// TIA Portal project "Template_ITIA2021" (V15.1)

(* hardware
DEVICE "S71500/ET200MP station_1"  S7-1500 station
   slot 0: "Rail_0"  Rack  6ES7 590-1***0-0AA0
   slot 0: "PM 70W 120/230VAC"  PM 70W 120/230VAC  6EP1332-4BA00
   slot 1: "Target_12_PLC"  CPU 1513-1 PN  6ES7 513-1AL02-0AB0  V2.6
      slot 3: "CPU display_1"  6ES7591-1AA00-0AA0
DEVICE "S71500/ET200MP station_2"  S7-1500 station
   slot 0: "Rail_0"  Rack  6ES7 590-1***0-0AA0
   slot 0: "PM 70W 120/230VAC"  PM 70W 120/230VAC  6EP1332-4BA00
   slot 1: "Target_34_PLC"  CPU 1513-1 PN  6ES7 513-1AL02-0AB0  V2.6
      slot 3: "CPU display_1"  6ES7591-1AA00-0AA0
DEVICE "S71500/ET200MP station_3"  S7-1500 station
   slot 0: "Rail_0"  Rack  6ES7 590-1***0-0AA0
   slot 0: "PM 70W 120/230VAC"  PM 70W 120/230VAC  6EP1332-4BA00
   slot 1: "Target_56_PLC"  CPU 1513-1 PN  6ES7 513-1AL02-0AB0  V2.6
      slot 3: "CPU display_1"  6ES7591-1AA00-0AA0
DEVICE "Target_12_HMI"  TP1500 Comfort
   slot 0: "Target_12_HMI"  TP1500 Comfort  6AV2 124-0QC02-0AX1  15.1.0.0
   slot 1: "HMI_RT_1"  TP1500 Comfort  6AV2 124-0QC02-0AX1  15.1.0.0
   slot 5: "Target_12_HMI.IE_CP_1"  PROFINET Interface  15.0.1.0
      slot 1: "PROFINET Interface_1"  PROFINET Interface
         slot 1: "Port_1"  Port
         slot 2: "Port_2"  Port
   slot 6: "Target_12_HMI.IE_CP_2"  PROFINET Interface  15.0.1.0
      slot 1: "PROFINET Interface_GBit"  PROFINET Interface
         slot 1: "Port_1"  Port
   slot 7: "Target_12_HMI.MPI/DP_CP_1"  MPI/DP Interface  15.0.1.0
DEVICE "SCALANCE X-200"  SCALANCE X-Station
   slot 0: "SCALANCE X rack"  Rail
   slot 0: "Target_12_Switch"  SCALANCE X208  6GK5 208-0BA00-2AA3  V1.0
DEVICE "SCALANCE X-200_1"  SCALANCE X-Station
   slot 0: "SCALANCE X rack"  Rail
   slot 0: "Target_34_Switch"  SCALANCE X208  6GK5 208-0BA00-2AA3  V1.0
DEVICE "SCALANCE X-200_2"  SCALANCE X-Station
   slot 0: "SCALANCE X rack"  Rail
   slot 0: "Target_56_Switch"  SCALANCE X208  6GK5 208-0BA00-2AA3  V1.0
DEVICE "ET 200SP station_1"  ET 200SP-Station
   slot 0: "Rack_0"  Rack  6ES5 710-8MAx1
   slot 0: "IO device_56"  IM 155-6 PN/2 HF  6ES7 155-6AU01-0CN0  V4.2
   slot 1: "CM AS-i Master ST_1"  CM AS-i Master ST  3RK7 137-6SA00-0BC1  V1.1
      slot 1: "CM AS-i Master ST"  CM AS-i Master ST
   slot 2: "DI 8x24VDC HF_1"  DI 8x24VDC HF  6ES7 131-6BF00-0CA0  V2.0
      slot 1: "DI 8x24VDC HF_1"  DI 8x24VDC HF
   slot 3: "DI 8x24VDC HF_2"  DI 8x24VDC HF  6ES7 131-6BF00-0CA0  V2.0
      slot 1: "DI 8x24VDC HF_2"  DI 8x24VDC HF
   slot 4: "DQ 8x24VDC/0.5A HF_1"  DQ 8x24VDC/0.5A HF  6ES7 132-6BF00-0CA0  V2.0
      slot 1: "DQ 8x24VDC/0.5A HF_1"  DQ 8x24VDC/0.5A HF
   slot 5: "DQ 8x24VDC/0.5A HF_2"  DQ 8x24VDC/0.5A HF  6ES7 132-6BF00-0CA0  V2.0
      slot 1: "DQ 8x24VDC/0.5A HF_2"  DQ 8x24VDC/0.5A HF
   slot 6: "Server module_1"  Server module  6ES7 193-6PA00-0AA0  V1.1
      slot 1: "Server module_1"  Server module
   slot 127: "BA 2xRJ45"  BA 2xRJ45  6ES7 193-6AR00-0AA0  V0.0
      slot 1: "Port_1"  X1 P1 R  6ES7 193-6AR00-0AA0  V0.0
      slot 2: "Port_2"  X1 P2 R  6ES7 193-6AR00-0AA0  V0.0
*)

// ===== PLC "Target_12_PLC"  CPU 1513-1 PN =====

ORGANIZATION_BLOCK "Main"   // OB1, LAD, ProgramCycle
TITLE = "Main Program Sweep (Cycle)"
{ S7_Optimized_Access := 'TRUE' }
VERSION : 0.1
   VAR_INPUT
      Initial_Call : Bool;   // Initial call of this OB
      Remanence : Bool;   // =True, if remanent data are available
   END_VAR
BEGIN
END_ORGANIZATION_BLOCK

// ===== PLC "Target_34_PLC"  CPU 1513-1 PN =====

ORGANIZATION_BLOCK "Main"   // OB1, LAD, ProgramCycle
TITLE = "Main Program Sweep (Cycle)"
{ S7_Optimized_Access := 'TRUE' }
VERSION : 0.1
   VAR_INPUT
      Initial_Call : Bool;   // Initial call of this OB
      Remanence : Bool;   // =True, if remanent data are available
   END_VAR
BEGIN
END_ORGANIZATION_BLOCK

// ===== PLC "Target_56_PLC"  CPU 1513-1 PN =====

VAR_GLOBAL   // PLC tag table "DefaultTable"
   "System_Byte" AT %MB1 : Byte;
   "FirstScan" AT %M1.0 : Bool;
   "DiagStatusUpdate" AT %M1.1 : Bool;
   "AlwaysTRUE" AT %M1.2 : Bool;
   "AlwaysFALSE" AT %M1.3 : Bool;
   "Clock_Byte" AT %MB0 : Byte;
   "Clock_10Hz" AT %M0.0 : Bool;
   "Clock_5Hz" AT %M0.1 : Bool;
   "Clock_2.5Hz" AT %M0.2 : Bool;
   "Clock_2Hz" AT %M0.3 : Bool;
   "Clock_1.25Hz" AT %M0.4 : Bool;
   "Clock_1Hz" AT %M0.5 : Bool;
   "Clock_0.625Hz" AT %M0.6 : Bool;
   "Clock_0.5Hz" AT %M0.7 : Bool;
END_VAR

VAR_GLOBAL   // PLC tag table "Station6"
   "S6_ButtonY" AT %I12.0 : Bool;
   "S6_ButtonG" AT %I12.1 : Bool;
   "S6_ButtonW" AT %I12.2 : Bool;
   "S6_ButtonR" AT %I12.3 : Bool;
   "S6_ItemInput_IsPresent" AT %I33.0 : Bool;
   "S6_Gate1_IsOpen" AT %I33.1 : Bool;
   "S6_Gate1_IsClosed" AT %I33.2 : Bool;
   "S6_Gate2_IsOpen" AT %I33.3 : Bool;
   "S6_ItemSlide_IsPresent" AT %I33.4 : Bool;
   "S6_Gate2_IsClosed" AT %I33.5 : Bool;
   "S6_LampY" AT %A12.0 : Bool;
   "S6_LampG" AT %Q12.1 : Bool;
   "S6_LampW" AT %Q12.2 : Bool;
   "S6_LampR" AT %Q12.3 : Bool;
   "S6_Belt_On" AT %Q33.0 : Bool;
   "S6_Gate2_Act" AT %Q14.4 : Bool;
   "S6_Gate1_Act" AT %Q14.5 : Bool;
   "S6_Stopper_Act" AT %Q14.6 : Bool;
END_VAR

VAR_GLOBAL   // PLC tag table "Station5"
   "S5_ButtonY" AT %E10.0 : Bool;
   "S5_ButtonG" AT %I10.1 : Bool;
   "S5_ButtonW" AT %I10.2 : Bool;
   "S5_ButtonR" AT %I10.3 : Bool;
   "S5_Cylinder_IsUp" AT %E32.0 : Bool;
   "S5_ItemMiddle_IsPresent" AT %I32.1 : Bool;
   "S5_ItemLeft_IsPresent" AT %I32.2 : Bool;
   "S5_Cylinder_IsDown" AT %I32.3 : Bool;
   "S5_ItemRight_IsPresent" AT %I32.4 : Bool;
   "S5_LampY" AT %A10.0 : Bool;
   "S5_LampG" AT %Q10.1 : Bool;
   "S5_LampW" AT %Q10.2 : Bool;
   "S5_LampR" AT %Q10.3 : Bool;
   "S5_SignalTowerG" AT %A11.4 : Bool;
   "S5_SignalTowerY" AT %Q11.5 : Bool;
   "S5_SignalTowerR" AT %A11.0 : Bool;
   "S5_Belt_On" AT %A32.0 : Bool;
   "S5_Cylinder_Act" AT %A12.4 : Bool;
   "request" AT %M2.0 : Bool;
   "ack" AT %M2.1 : Bool;
   "material" AT %MW1 : UInt;
   "emergency_stop" AT %M2.3 : Bool;
END_VAR

// folder: SystemDataTypeFolder

TYPE "Client interface_target1.Read list_target1"
   STRUCT
      Emergency_S1 : Bool;
      Error_S1 : Bool;
      Running_S1 : Bool;
      Emergency_S2 : Bool;
      Error_S2 : Bool;
      Running_S2 : Bool;
      Tower_emptey_S1 : Bool;
   END_STRUCT;
END_TYPE

TYPE "Client interface_target3.Read list_target3"
   STRUCT
      request : Bool;
      material : USInt;
      Emergency_S3 : Bool;
      Running_S3 : Bool;
   END_STRUCT;
END_TYPE

// folder: (top level)

DATA_BLOCK "Station5_DB"   // DB1
{ S7_Optimized_Access := 'TRUE' }
VERSION : 0.1
// stored: InstanceOfName Station5
"Station5"
BEGIN
END_DATA_BLOCK

DATA_BLOCK "Station6_DB"   // DB2
{ S7_Optimized_Access := 'TRUE' }
VERSION : 0.1
// stored: InstanceOfName Station6
"Station6"
BEGIN
END_DATA_BLOCK

DATA_BLOCK "ServerVariables_DB"   // DB3
{ S7_Optimized_Access := 'TRUE' }
VERSION : 0.1
   VAR
      emergency_stop : Bool;
      material : Byte;
      request : Bool;
      Emergency_Stop_S5 : Bool;
      Reset_S5 : Bool;
      Start_S5 : Bool;
      Emergency_S6 : Bool;
      Running_S6 : Bool;
      Error_S6 : Bool;
      Emergency_S5 : Bool;
      Running_S5 : Bool;
      Error_S5 : Bool;
      ack : Bool;
   END_VAR
BEGIN
END_DATA_BLOCK

DATA_BLOCK "Client interface_target3_Data"   // DB5
{ S7_Optimized_Access := 'TRUE' }
VERSION : 0.1
   VAR
      "Read list_target3" : Struct
         Variable : "Client interface_target3.Read list_target3";
         NodeStatusList : Array[0..3] of DWord;
         TimeStamps : Array[0..3] of LDT;
      END_STRUCT;
   END_VAR
BEGIN
END_DATA_BLOCK

DATA_BLOCK "Client interface_target1_Data"   // DB11
{ S7_Optimized_Access := 'TRUE' }
VERSION : 0.1
   VAR
      "Read list_target1" : Struct
         Variable : "Client interface_target1.Read list_target1";
         NodeStatusList : Array[0..6] of DWord;
         TimeStamps : Array[0..6] of LDT;
      END_STRUCT;
   END_VAR
BEGIN
END_DATA_BLOCK

DATA_BLOCK "Client_interface_target1_DB"   // DB16
{ S7_Optimized_Access := 'TRUE' }
VERSION : 0.1
// stored: InstanceOfName Client_interface_target1
"Client_interface_target1"
BEGIN
END_DATA_BLOCK

DATA_BLOCK "Client_interface_target3_DB"   // DB17
{ S7_Optimized_Access := 'TRUE' }
VERSION : 0.1
// stored: InstanceOfName Client_interface_target3
"Client_interface_target3"
BEGIN
END_DATA_BLOCK

DATA_BLOCK "FIFO_DB"   // DB20
{ S7_Optimized_Access := 'TRUE' }
VERSION : 0.1
// stored: InstanceOfName FIFO
"FIFO"
BEGIN
END_DATA_BLOCK

// folder: System blocks/Program resources

DATA_BLOCK "Client interface_target3_Configuration"   // DB4
{ S7_Optimized_Access := 'TRUE' }
VERSION : 0.1
   VAR
      Connection : Struct
         ConnectInfo : OPC_UA_SessionConnectInfo;
         ConnectionHdl : DWord;
         ServerEndpointUrl : String[254] := 'opc.tcp://192.168.162.49:4840';
      END_STRUCT;
      Namespaces : Struct
         NamespaceURIs : Array[0..0] of WString;
         ServerNamespaceIndexes : Array[0..0] of UInt;
         NamespaceStatusList : Array[0..0] of DWord;
         NamespaceCount : UInt := 1;
      END_STRUCT;
      ReadLists : Struct
         "Read list_target3" : Struct
            NodeCount : UInt := 4;
            Nodes : Array[0..3] of OPC_UA_NodeId;
            NodeHdls : Array[0..3] of DWord;
         END_STRUCT;
      END_STRUCT;
   END_VAR
BEGIN
   ReadLists."Read list_target3".Nodes[0].NamespaceIndex := 0;
   ReadLists."Read list_target3".Nodes[0].IdentifierType := 0;
   ReadLists."Read list_target3".Nodes[0].Identifier := WSTRING#'6011';
   ReadLists."Read list_target3".Nodes[1].NamespaceIndex := 0;
   ReadLists."Read list_target3".Nodes[1].IdentifierType := 0;
   ReadLists."Read list_target3".Nodes[1].Identifier := WSTRING#'6013';
   ReadLists."Read list_target3".Nodes[2].NamespaceIndex := 0;
   ReadLists."Read list_target3".Nodes[2].IdentifierType := 0;
   ReadLists."Read list_target3".Nodes[2].Identifier := WSTRING#'6008';
   ReadLists."Read list_target3".Nodes[3].NamespaceIndex := 0;
   ReadLists."Read list_target3".Nodes[3].IdentifierType := 0;
   ReadLists."Read list_target3".Nodes[3].Identifier := WSTRING#'6009';
   Connection.ConnectInfo.SessionName := WSTRING#'OPC UA Connection_1';
   Connection.ConnectInfo.ApplicationName := WSTRING#'';
   Connection.ConnectInfo.SecurityMsgMode := 1;
   Connection.ConnectInfo.SecurityPolicy := 1;
   Connection.ConnectInfo.ServerUri := '';
   Connection.ConnectInfo.CheckServerCertificate := False;
   Connection.ConnectInfo.TransportProfile := 1;
   Connection.ConnectInfo.UserIdentityTokenType := 0;
   Connection.ConnectInfo.CertificateID := 0;
   Connection.ConnectInfo.SessionTimeout := T#30S;
   Connection.ConnectInfo.MonitorConnection := T#5S;
   Connection.ConnectInfo.LocaleIDs[0] := 'en-US';
   Connection.ConnectInfo.LocaleIDs[1] := '';
   Connection.ConnectInfo.LocaleIDs[2] := '';
   Connection.ConnectInfo.LocaleIDs[3] := '';
   Connection.ConnectInfo.LocaleIDs[4] := '';
   Namespaces.NamespaceURIs[0] := WSTRING#'http://itia_target_2';
END_DATA_BLOCK

DATA_BLOCK "Client interface_target1_Configuration"   // DB10
{ S7_Optimized_Access := 'TRUE' }
VERSION : 0.1
   VAR
      Connection : Struct
         ConnectInfo : OPC_UA_SessionConnectInfo;
         ConnectionHdl : DWord;
         ServerEndpointUrl : String[254] := 'opc.tcp://192.168.162.33:4840';
      END_STRUCT;
      Namespaces : Struct
         NamespaceURIs : Array[0..0] of WString;
         ServerNamespaceIndexes : Array[0..0] of UInt;
         NamespaceStatusList : Array[0..0] of DWord;
         NamespaceCount : UInt := 1;
      END_STRUCT;
      ReadLists : Struct
         "Read list_target1" : Struct
            NodeCount : UInt := 7;
            Nodes : Array[0..6] of OPC_UA_NodeId;
            NodeHdls : Array[0..6] of DWord;
         END_STRUCT;
      END_STRUCT;
   END_VAR
BEGIN
   ReadLists."Read list_target1".Nodes[0].NamespaceIndex := 0;
   ReadLists."Read list_target1".Nodes[0].IdentifierType := 0;
   ReadLists."Read list_target1".Nodes[0].Identifier := WSTRING#'6010';
   ReadLists."Read list_target1".Nodes[1].NamespaceIndex := 0;
   ReadLists."Read list_target1".Nodes[1].IdentifierType := 0;
   ReadLists."Read list_target1".Nodes[1].Identifier := WSTRING#'6021';
   ReadLists."Read list_target1".Nodes[2].NamespaceIndex := 0;
   ReadLists."Read list_target1".Nodes[2].IdentifierType := 0;
   ReadLists."Read list_target1".Nodes[2].Identifier := WSTRING#'6022';
   ReadLists."Read list_target1".Nodes[3].NamespaceIndex := 0;
   ReadLists."Read list_target1".Nodes[3].IdentifierType := 0;
   ReadLists."Read list_target1".Nodes[3].Identifier := WSTRING#'6011';
   ReadLists."Read list_target1".Nodes[4].NamespaceIndex := 0;
   ReadLists."Read list_target1".Nodes[4].IdentifierType := 0;
   ReadLists."Read list_target1".Nodes[4].Identifier := WSTRING#'6023';
   ReadLists."Read list_target1".Nodes[5].NamespaceIndex := 0;
   ReadLists."Read list_target1".Nodes[5].IdentifierType := 0;
   ReadLists."Read list_target1".Nodes[5].Identifier := WSTRING#'6024';
   ReadLists."Read list_target1".Nodes[6].NamespaceIndex := 0;
   ReadLists."Read list_target1".Nodes[6].IdentifierType := 0;
   ReadLists."Read list_target1".Nodes[6].Identifier := WSTRING#'6012';
   Connection.ConnectInfo.SessionName := WSTRING#'OPC UA Connection_1';
   Connection.ConnectInfo.ApplicationName := WSTRING#'';
   Connection.ConnectInfo.SecurityMsgMode := 1;
   Connection.ConnectInfo.SecurityPolicy := 1;
   Connection.ConnectInfo.ServerUri := '';
   Connection.ConnectInfo.CheckServerCertificate := False;
   Connection.ConnectInfo.TransportProfile := 1;
   Connection.ConnectInfo.UserIdentityTokenType := 0;
   Connection.ConnectInfo.CertificateID := 0;
   Connection.ConnectInfo.SessionTimeout := T#30S;
   Connection.ConnectInfo.MonitorConnection := T#5S;
   Connection.ConnectInfo.LocaleIDs[0] := 'en-US';
   Connection.ConnectInfo.LocaleIDs[1] := '';
   Connection.ConnectInfo.LocaleIDs[2] := '';
   Connection.ConnectInfo.LocaleIDs[3] := '';
   Connection.ConnectInfo.LocaleIDs[4] := '';
   Namespaces.NamespaceURIs[0] := WSTRING#'http://tia_target1';
END_DATA_BLOCK

DATA_BLOCK "IEC_Timer_0_DB"   // DB21
{ S7_Optimized_Access := 'TRUE' }
AUTHOR : Simatic
FAMILY : IEC
NAME : IEC_TMR
VERSION : 1.0
// stored: InstanceOfName IEC_TIMER
"IEC_TIMER"
BEGIN
END_DATA_BLOCK

DATA_BLOCK "IEC_Timer_0_DB_1"   // DB22
{ S7_Optimized_Access := 'TRUE' }
AUTHOR : Simatic
FAMILY : IEC
NAME : IEC_TMR
VERSION : 1.0
// stored: InstanceOfName IEC_TIMER
"IEC_TIMER"
BEGIN
END_DATA_BLOCK

// folder: (top level)

FUNCTION_BLOCK "Station5"   // FB1, FBD
TITLE = Station5
{ S7_Optimized_Access := 'TRUE' }
VERSION : 0.1
   VAR_INPUT
      station6_ack : Bool;
      slide_full : Bool;
      material_in : Int;
      global_error : Bool;
      station6_sorting_done : Bool;
      station4_req : Bool;
   END_VAR
   VAR_OUTPUT
      global_error_out : Bool;
      station5_req : Bool;
      station5_ack : Bool;
      material_out : Int := 1;
      belt_start : Bool := false;
   END_VAR
   VAR
      STOP : Bool;
      belt_on_var : Bool;
      workpiece_arr_pos : UInt;
      station4_ack_occurred : Bool;
      work : Bool;
      count_workpieces : UInt;
      place_no_further_working_piece : Bool;
      workpiece_found_middle : Bool;
      reset_cyclinder : Bool;
      emergency_client_S1 : Bool;
      ERROR : Bool;
      RUNNING : Bool;
      EMERGENCY : Bool;
      station6_ack_occured : Bool;
      workpiece_could_pass : Bool;
      fifo_buffer_full : Bool;
      fifo_buffer_empty : Bool;
      fifo_data_out : Int;
      left_trigger : Bool;
      right_trigger : Bool;
      stop_belt : Bool;
      materialFrom4 : UInt;
      emergency_occured : Bool;
      error_occured : Bool;
      set_tower_red : Bool;
   END_VAR
   VAR_TEMP   // added for the SCL form of the ladder/FBD networks
      _w1 : Bool;
      _w2 : Bool;
      _w3 : Bool;
   END_VAR
BEGIN

REGION Network 1: Initial call of this FB
   // error + starting, extended logic for running and emergency mode regarding the opc ua communication
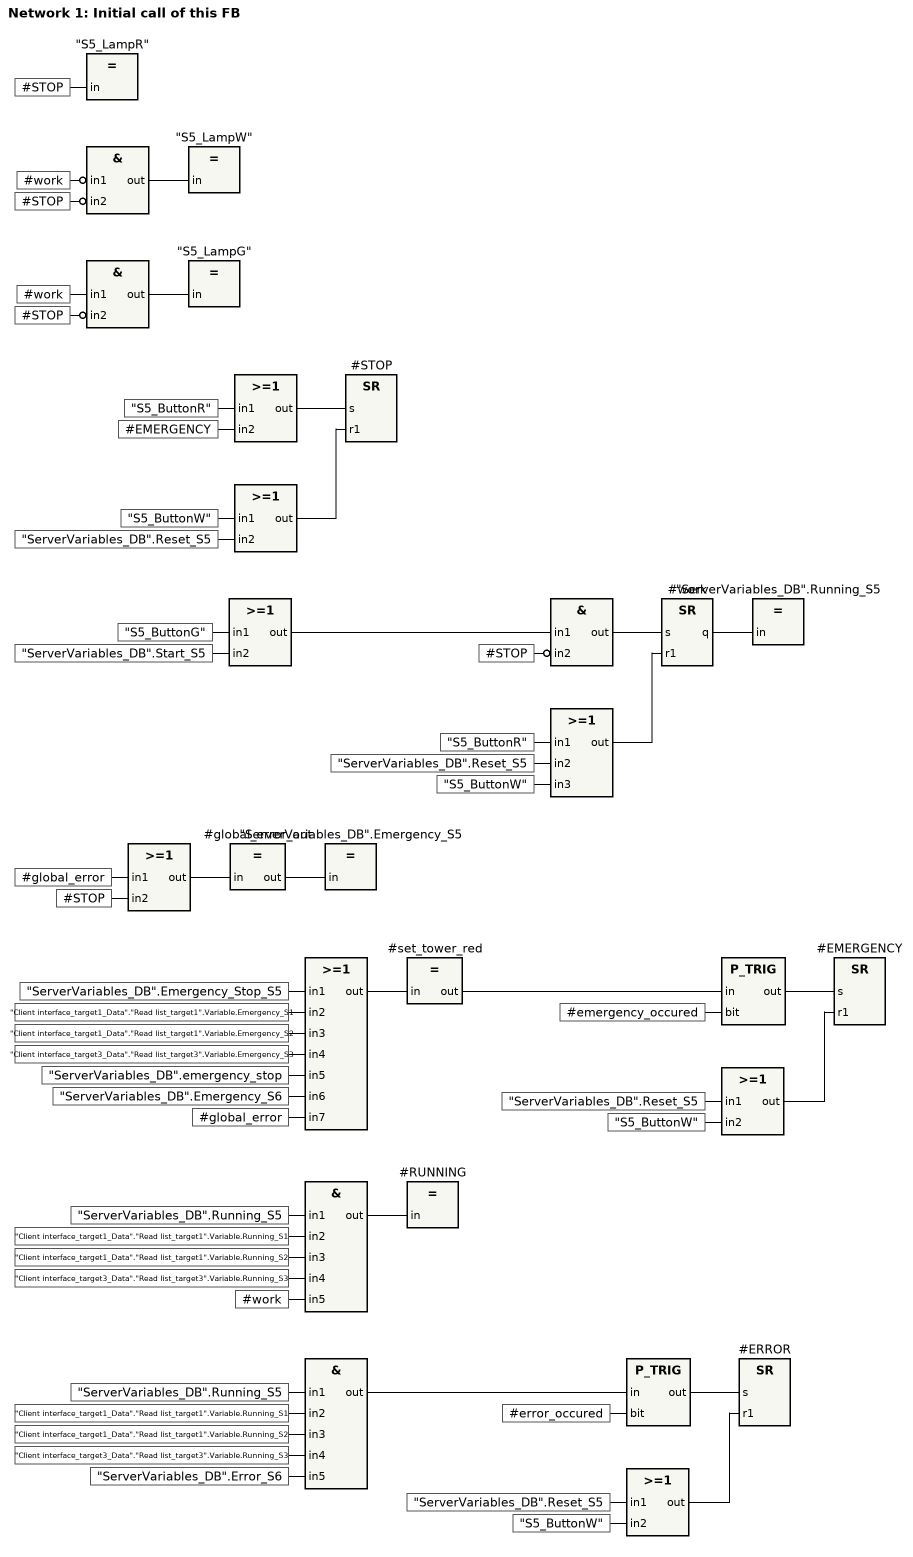
   "S5_LampR" := #STOP;
   "S5_LampW" := NOT #work AND NOT #STOP;
   "S5_LampG" := #work AND NOT #STOP;
   IF "S5_ButtonR" OR #EMERGENCY THEN
       #STOP := TRUE;   // SR flip-flop
   END_IF;
   IF "S5_ButtonW" OR "ServerVariables_DB".Reset_S5 THEN #STOP := FALSE; END_IF;
   IF ("S5_ButtonG" OR "ServerVariables_DB".Start_S5) AND NOT #STOP THEN
       #work := TRUE;   // SR flip-flop
   END_IF;
   IF "S5_ButtonR" OR "ServerVariables_DB".Reset_S5 OR "S5_ButtonW" THEN #work := FALSE; END_IF;
   "ServerVariables_DB".Running_S5 := #work;
   #global_error_out := #global_error OR #STOP;
   "ServerVariables_DB".Emergency_S5 := #global_error_out;
   #set_tower_red := "ServerVariables_DB".Emergency_Stop_S5 OR "Client interface_target1_Data"."Read list_target1".Variable.Emergency_S1 OR "Client interface_target1_Data"."Read list_target1".Variable.Emergency_S2 OR "Client interface_target3_Data"."Read list_target3".Variable.Emergency_S3 OR "ServerVariables_DB".emergency_stop OR "ServerVariables_DB".Emergency_S6 OR #global_error;
   #_w1 := #set_tower_red AND NOT #emergency_occured;   // rising edge
   #emergency_occured := #set_tower_red;
   IF #_w1 THEN
       #EMERGENCY := TRUE;   // SR flip-flop
   END_IF;
   IF "ServerVariables_DB".Reset_S5 OR "S5_ButtonW" THEN #EMERGENCY := FALSE; END_IF;
   #RUNNING := "ServerVariables_DB".Running_S5 AND "Client interface_target1_Data"."Read list_target1".Variable.Running_S1 AND "Client interface_target1_Data"."Read list_target1".Variable.Running_S2 AND "Client interface_target3_Data"."Read list_target3".Variable.Running_S3 AND #work;
   #_w2 := "ServerVariables_DB".Running_S5 AND "Client interface_target1_Data"."Read list_target1".Variable.Running_S1 AND "Client interface_target1_Data"."Read list_target1".Variable.Running_S2 AND "Client interface_target3_Data"."Read list_target3".Variable.Running_S3 AND "ServerVariables_DB".Error_S6;
   #_w3 := #_w2 AND NOT #error_occured;   // rising edge
   #error_occured := #_w2;
   IF #_w3 THEN
       #ERROR := TRUE;   // SR flip-flop
   END_IF;
   IF "ServerVariables_DB".Reset_S5 OR "S5_ButtonW" THEN #ERROR := FALSE; END_IF;
END_REGION

REGION Network 2: Belt movement
   // Move belt when workmode is on, stop it when station 4 request is acknowledged or while waiting for station 6 ack
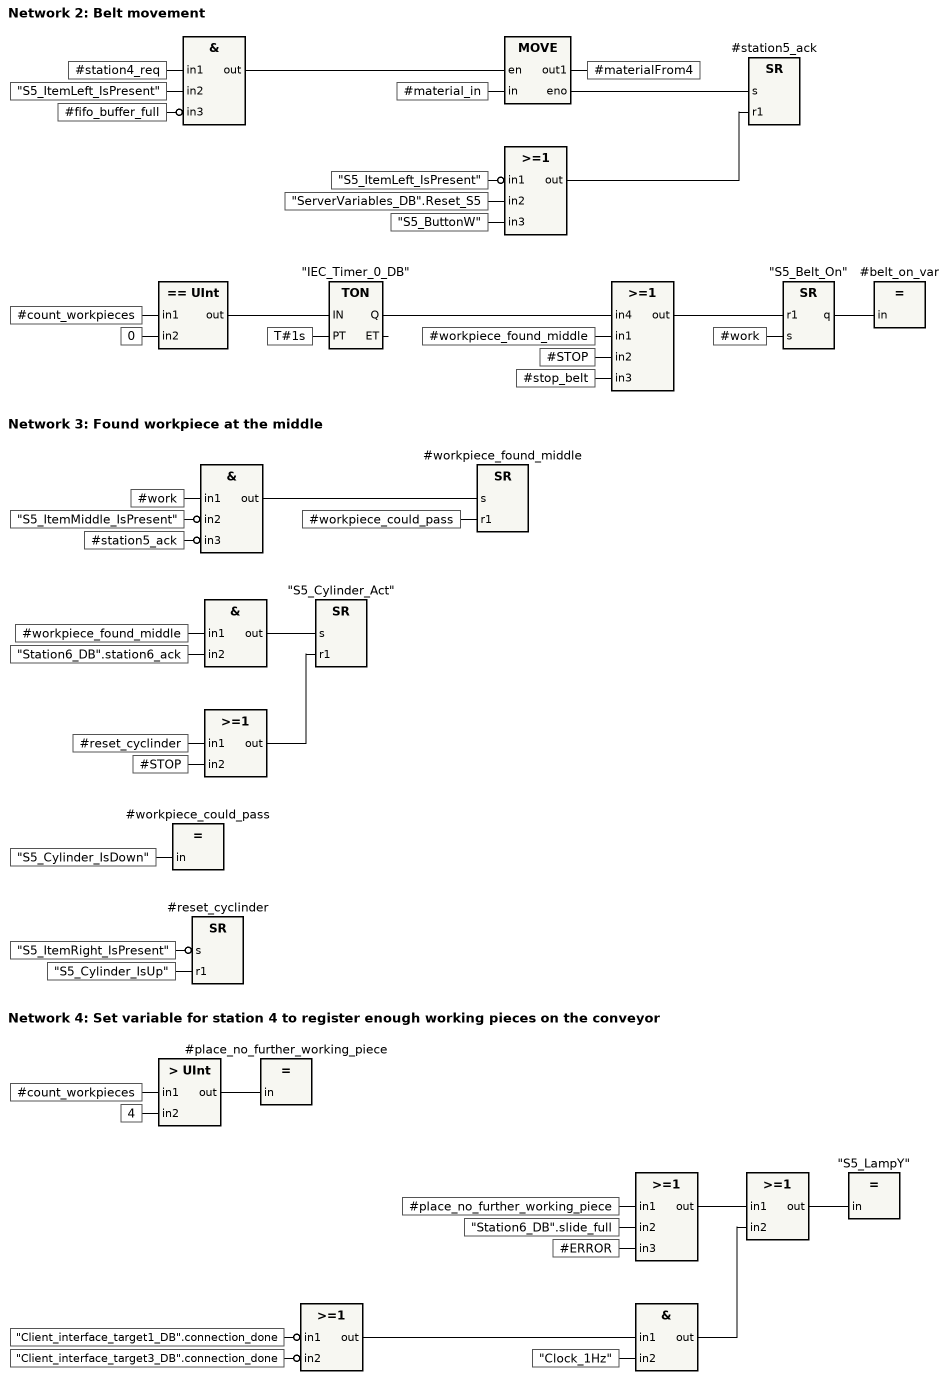
   #_w1 := #station4_req AND "S5_ItemLeft_IsPresent" AND NOT #fifo_buffer_full;
   IF #_w1 THEN
       #materialFrom4 := #material_in;
       #station5_ack := TRUE;   // SR flip-flop
   END_IF;
   IF NOT "S5_ItemLeft_IsPresent" OR "ServerVariables_DB".Reset_S5 OR "S5_ButtonW" THEN
       #station5_ack := FALSE;
   END_IF;
   "IEC_Timer_0_DB".TON(IN := #count_workpieces = 0, PT := T#1s);
   IF #work THEN
       "S5_Belt_On" := TRUE;   // SR flip-flop
   END_IF;
   IF "IEC_Timer_0_DB".Q OR #workpiece_found_middle OR #STOP OR #stop_belt THEN
       "S5_Belt_On" := FALSE;
   END_IF;
   #belt_on_var := "S5_Belt_On";
END_REGION

REGION Network 3: Found workpiece at the middle
   // workflow of cylinder
   IF #work AND NOT "S5_ItemMiddle_IsPresent" AND NOT #station5_ack THEN
       #workpiece_found_middle := TRUE;   // SR flip-flop
   END_IF;
   IF #workpiece_could_pass THEN #workpiece_found_middle := FALSE; END_IF;
   IF #workpiece_found_middle AND "Station6_DB".station6_ack THEN
       "S5_Cylinder_Act" := TRUE;   // SR flip-flop
   END_IF;
   IF #reset_cyclinder OR #STOP THEN "S5_Cylinder_Act" := FALSE; END_IF;
   #workpiece_could_pass := "S5_Cylinder_IsDown";
   IF NOT "S5_ItemRight_IsPresent" THEN
       #reset_cyclinder := TRUE;   // SR flip-flop
   END_IF;
   IF "S5_Cylinder_IsUp" THEN #reset_cyclinder := FALSE; END_IF;
END_REGION

REGION Network 4: Set variable for station 4 to register enough working pieces on the conveyor
   // Interface with station 4 and 6
   #place_no_further_working_piece := #count_workpieces > 4;
   "S5_LampY" := #place_no_further_working_piece OR "Station6_DB".slide_full OR #ERROR OR ((NOT "Client_interface_target1_DB".connection_done OR NOT "Client_interface_target3_DB".connection_done) AND "Clock_1Hz");
END_REGION

REGION Network 5: Counter for workpiece check if buffer full
   // Counter needed to check if station 4 could place workpiece
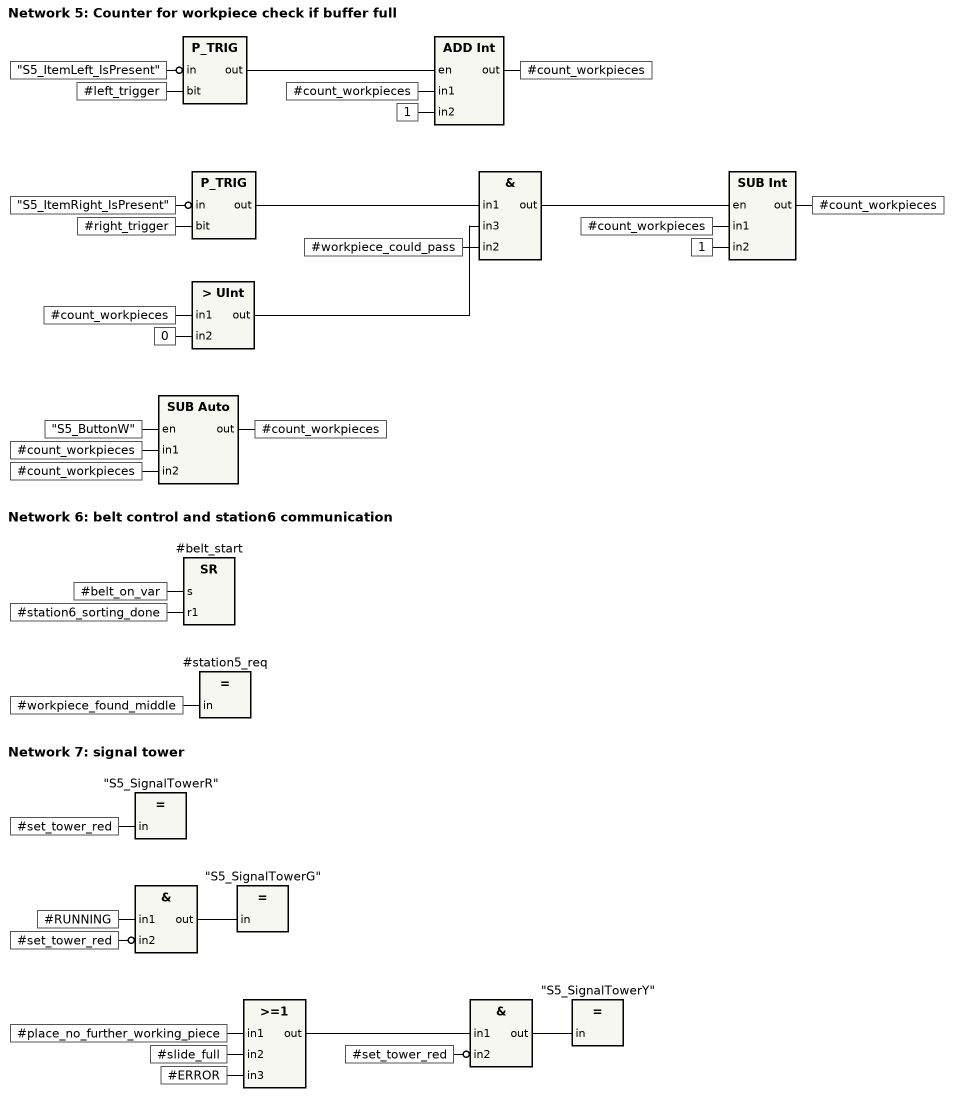
   #_w1 := NOT "S5_ItemLeft_IsPresent" AND NOT #left_trigger;   // rising edge
   #left_trigger := NOT "S5_ItemLeft_IsPresent";
   IF #_w1 THEN #count_workpieces := #count_workpieces + 1; END_IF;
   #_w2 := NOT "S5_ItemRight_IsPresent" AND NOT #right_trigger;   // rising edge
   #right_trigger := NOT "S5_ItemRight_IsPresent";
   IF #_w2 AND (#count_workpieces > 0) AND #workpiece_could_pass THEN
       #count_workpieces := #count_workpieces - 1;
   END_IF;
   IF "S5_ButtonW" THEN #count_workpieces := #count_workpieces - #count_workpieces; END_IF;
END_REGION

REGION Network 6: belt control and station6 communication
   // Interface station 6 communication
   // send material info to station 6
   IF #belt_on_var THEN
       #belt_start := TRUE;   // SR flip-flop
   END_IF;
   IF #station6_sorting_done THEN #belt_start := FALSE; END_IF;
   #station5_req := #workpiece_found_middle;
END_REGION

REGION Network 7: signal tower
   // Tower lamps using the overall plant signals of the OPC UA communication and the intern signal to represent a 'global' status
   "S5_SignalTowerR" := #set_tower_red;
   "S5_SignalTowerG" := #RUNNING AND NOT #set_tower_red;
   "S5_SignalTowerY" := (#place_no_further_working_piece OR #slide_full OR #ERROR) AND NOT #set_tower_red;
END_REGION

REGION Network 8
   // Interface variables has to be checked if an emergency occured there (set the status of the emergency of station 5 itself)
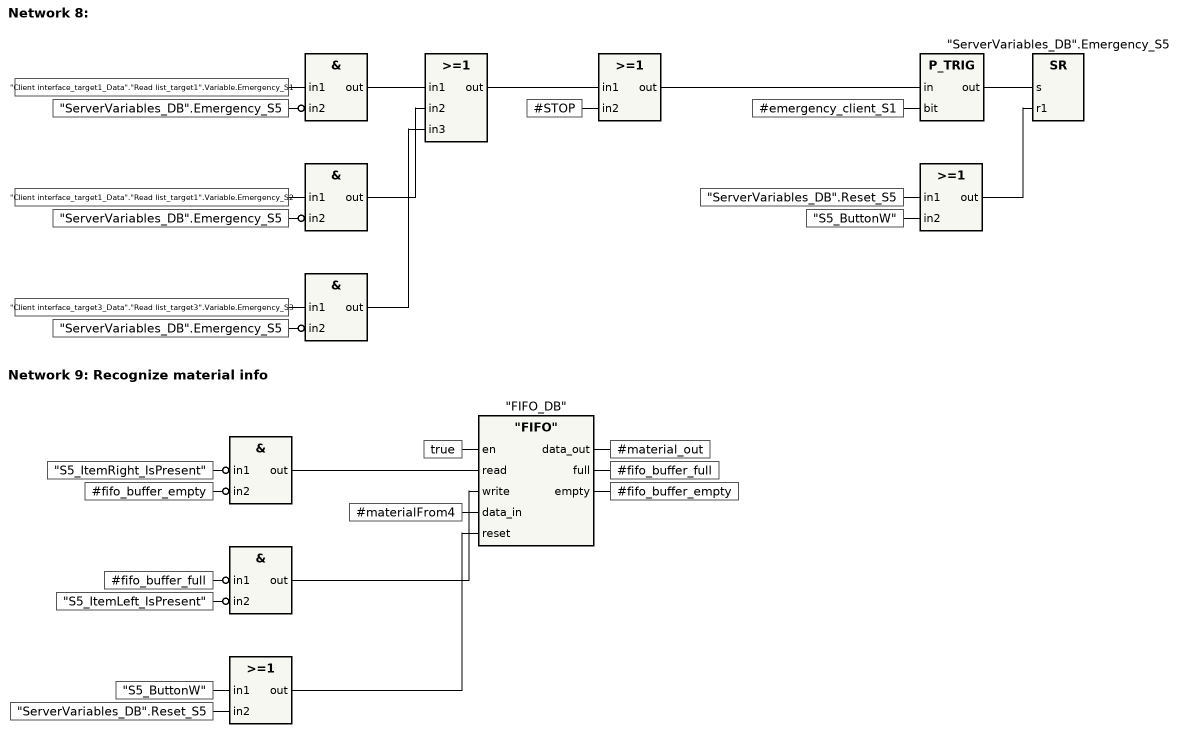
   #_w1 := ("Client interface_target1_Data"."Read list_target1".Variable.Emergency_S1 AND NOT "ServerVariables_DB".Emergency_S5) OR ("Client interface_target1_Data"."Read list_target1".Variable.Emergency_S2 AND NOT "ServerVariables_DB".Emergency_S5) OR ("Client interface_target3_Data"."Read list_target3".Variable.Emergency_S3 AND NOT "ServerVariables_DB".Emergency_S5) OR #STOP;
   #_w2 := #_w1 AND NOT #emergency_client_S1;   // rising edge
   #emergency_client_S1 := #_w1;
   IF #_w2 THEN
       "ServerVariables_DB".Emergency_S5 := TRUE;   // SR flip-flop
   END_IF;
   IF "ServerVariables_DB".Reset_S5 OR "S5_ButtonW" THEN "ServerVariables_DB".Emergency_S5 := FALSE; END_IF;
END_REGION

REGION Network 9: Recognize material info
   // use the FIFO buffer to store specific material info and forward it to station 6
   IF true THEN
       "FIFO_DB"(read := NOT "S5_ItemRight_IsPresent" AND NOT #fifo_buffer_empty,   // "FIFO"
                 write := NOT #fifo_buffer_full AND NOT "S5_ItemLeft_IsPresent",
                 data_in := #materialFrom4,
                 reset := "S5_ButtonW" OR "ServerVariables_DB".Reset_S5,
                 data_out => #material_out,
                 full => #fifo_buffer_full,
                 empty => #fifo_buffer_empty);
   END_IF;
END_REGION
END_FUNCTION_BLOCK

FUNCTION_BLOCK "Station6"   // FB2, FBD
TITLE = Station6
{ S7_Optimized_Access := 'TRUE' }
VERSION : 0.1
   VAR_INPUT
      station5_req : Bool;
      material_in : UInt;
      global_error : Bool;
      belt_start : Bool;
   END_VAR
   VAR_OUTPUT
      station6_ack : Bool;
      sorting_done : Bool;
      slide_full : Bool;
   END_VAR
   VAR
      STOP : Bool;
      init : Bool;
      running : Bool;
      inputReady : Bool;
      startSort : Bool;
      waitForSortingDone : Bool;
      piecePassedSlide : Bool;
      presentTimeout : Bool;
      ItemSlideNotPresent : Bool;
      slideFullDelayer : IEC_TIMER;
      ready_to_sort : Bool;
      request_occured : Bool;
      sortMaterial : UInt;
      glob_error_s5 : Bool;
      slide_full_delayer : Bool;
   END_VAR
   VAR_TEMP   // added for the SCL form of the ladder/FBD networks
      _w1 : Bool;
      _w2 : Bool;
   END_VAR
BEGIN

REGION Network 1: activation & error handling
   // activate and init station6; reset error (STOP)
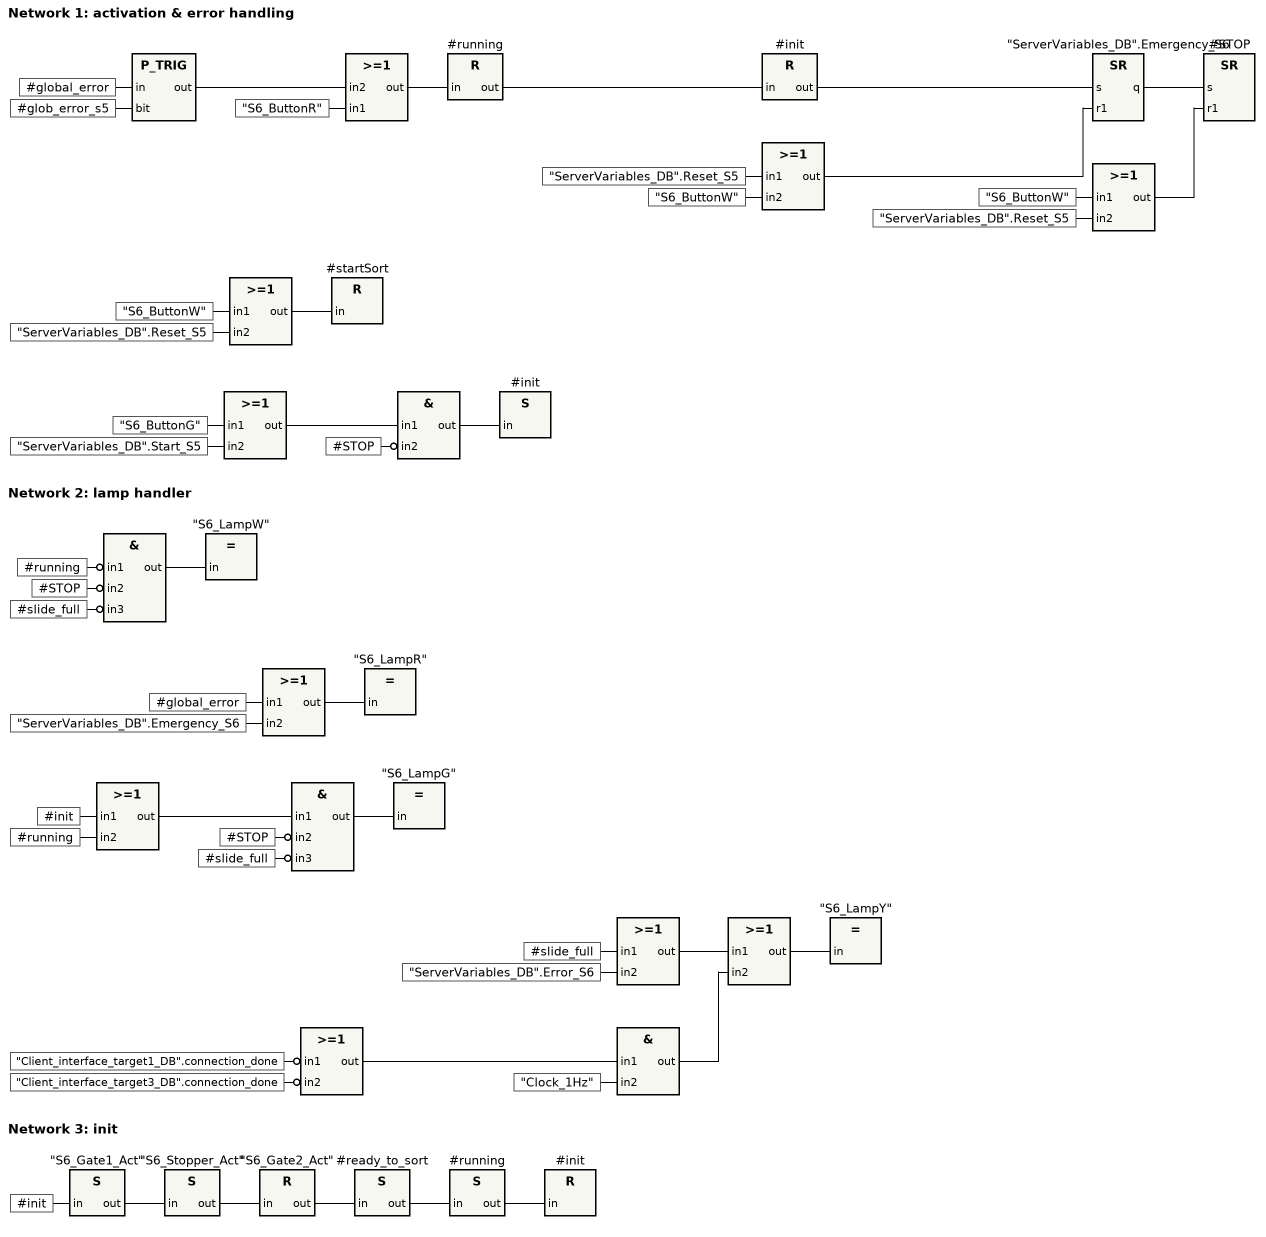
   #_w1 := #global_error AND NOT #glob_error_s5;   // rising edge
   #glob_error_s5 := #global_error;
   #_w2 := #_w1 OR "S6_ButtonR";
   IF #_w2 THEN
       #running := FALSE;
       #init := FALSE;
       "ServerVariables_DB".Emergency_S6 := TRUE;   // SR flip-flop
   END_IF;
   IF "ServerVariables_DB".Reset_S5 OR "S6_ButtonW" THEN "ServerVariables_DB".Emergency_S6 := FALSE; END_IF;
   IF "ServerVariables_DB".Emergency_S6 THEN
       #STOP := TRUE;   // SR flip-flop
   END_IF;
   IF "S6_ButtonW" OR "ServerVariables_DB".Reset_S5 THEN
       #STOP := FALSE;
       #startSort := FALSE;
   END_IF;
   IF ("S6_ButtonG" OR "ServerVariables_DB".Start_S5) AND NOT #STOP THEN #init := TRUE; END_IF;
END_REGION

REGION Network 2: lamp handler
   // white if ready to start; red if STOP(error); green if running basically and yellow if one slide barrier is broken for a long time ( = assuming full slide)
   "S6_LampW" := NOT #running AND NOT #STOP AND NOT #slide_full;
   "S6_LampR" := #global_error OR "ServerVariables_DB".Emergency_S6;
   "S6_LampG" := (#init OR #running) AND NOT #STOP AND NOT #slide_full;
   "S6_LampY" := #slide_full OR "ServerVariables_DB".Error_S6 OR ((NOT "Client_interface_target1_DB".connection_done OR NOT "Client_interface_target3_DB".connection_done) AND "Clock_1Hz");
END_REGION

REGION Network 3: init
   // init: gate1 closed,  gate2 open, Stopper extracted
   IF #init THEN
       "S6_Gate1_Act" := TRUE;
       "S6_Stopper_Act" := TRUE;
       "S6_Gate2_Act" := FALSE;
       #ready_to_sort := TRUE;
       #running := TRUE;
       #init := FALSE;
   END_IF;
END_REGION

REGION Network 4: handshake & start sort logic
   // sotre incoming material in variable on request; after request excpect material to actually come in and set variable to start the sorting
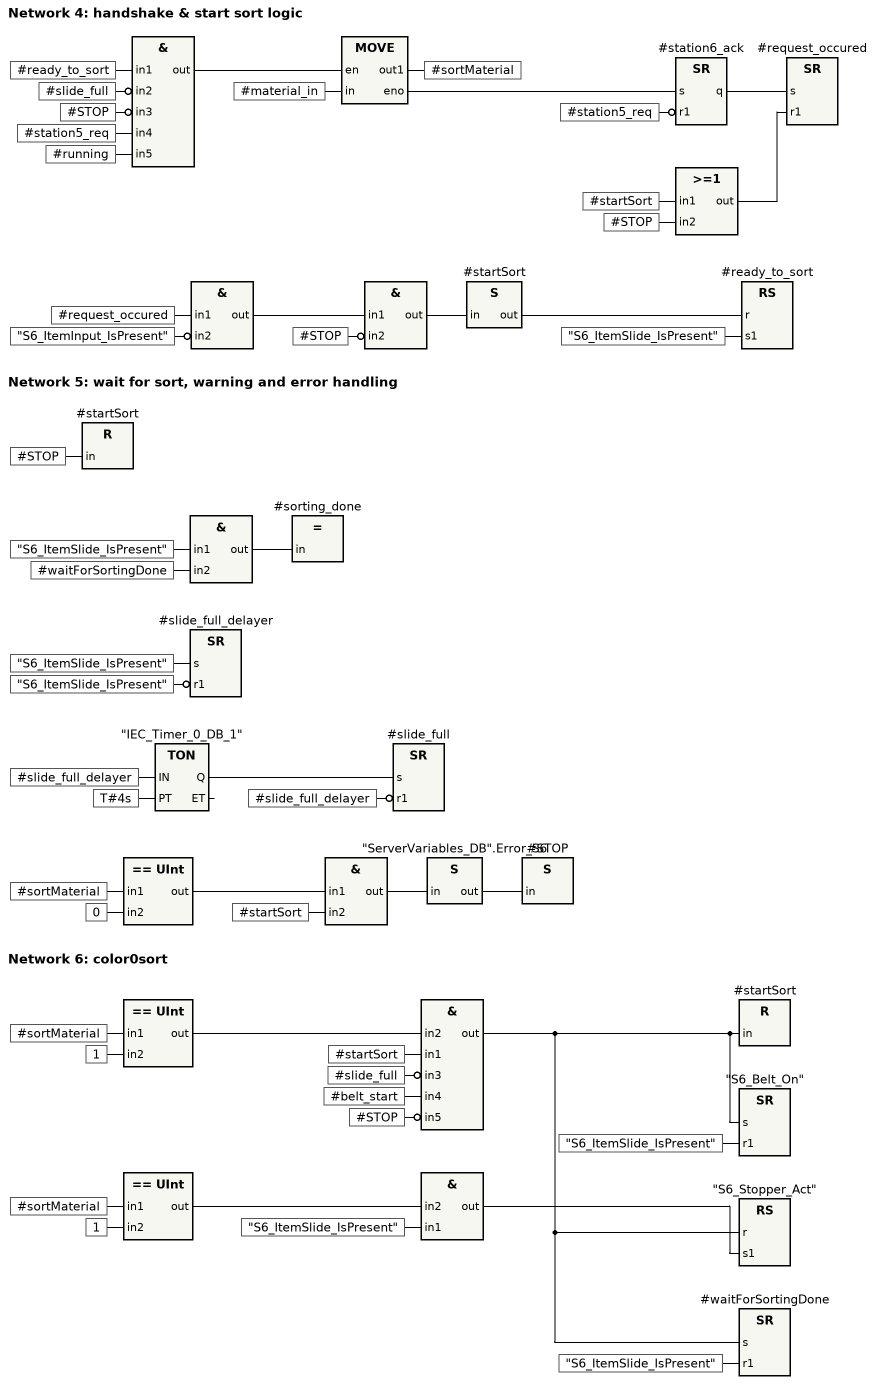
   #_w1 := #ready_to_sort AND NOT #slide_full AND NOT #STOP AND #station5_req AND #running;
   IF #_w1 THEN
       #sortMaterial := #material_in;
       #station6_ack := TRUE;   // SR flip-flop
   END_IF;
   IF NOT #station5_req THEN #station6_ack := FALSE; END_IF;
   IF #station6_ack THEN
       #request_occured := TRUE;   // SR flip-flop
   END_IF;
   IF #startSort OR #STOP THEN #request_occured := FALSE; END_IF;
   #_w2 := #request_occured AND NOT "S6_ItemInput_IsPresent" AND NOT #STOP;
   IF #_w2 THEN
       #startSort := TRUE;
       #ready_to_sort := FALSE;   // RS flip-flop
   END_IF;
   IF "S6_ItemSlide_IsPresent" THEN #ready_to_sort := TRUE; END_IF;
END_REGION

REGION Network 5: wait for sort, warning and error handling
   // sorting is done when something entered the slide; stop everything when stop flag is set
   IF #STOP THEN #startSort := FALSE; END_IF;
   #sorting_done := "S6_ItemSlide_IsPresent" AND #waitForSortingDone;
   IF "S6_ItemSlide_IsPresent" THEN
       #slide_full_delayer := TRUE;   // SR flip-flop
   END_IF;
   IF NOT "S6_ItemSlide_IsPresent" THEN #slide_full_delayer := FALSE; END_IF;
   "IEC_Timer_0_DB_1".TON(IN := #slide_full_delayer, PT := T#4s);
   IF "IEC_Timer_0_DB_1".Q THEN
       #slide_full := TRUE;   // SR flip-flop
   END_IF;
   IF NOT #slide_full_delayer THEN #slide_full := FALSE; END_IF;
   IF (#sortMaterial = 0) AND #startSort THEN
       "ServerVariables_DB".Error_S6 := TRUE;
       #STOP := TRUE;
   END_IF;
END_REGION

REGION Network 6: color0sort
   // sort color 0
   #_w1 := (#sortMaterial = 1) AND #startSort AND NOT #slide_full AND #belt_start AND NOT #STOP;
   IF #_w1 THEN
       #startSort := FALSE;
       "S6_Belt_On" := TRUE;   // SR flip-flop
   END_IF;
   IF "S6_ItemSlide_IsPresent" THEN "S6_Belt_On" := FALSE; END_IF;
   IF #_w1 THEN
       "S6_Stopper_Act" := FALSE;   // RS flip-flop
   END_IF;
   IF (#sortMaterial = 1) AND "S6_ItemSlide_IsPresent" THEN "S6_Stopper_Act" := TRUE; END_IF;
   IF #_w1 THEN
       #waitForSortingDone := TRUE;   // SR flip-flop
   END_IF;
   IF "S6_ItemSlide_IsPresent" THEN #waitForSortingDone := FALSE; END_IF;
END_REGION

REGION Network 7: color1sort
   // sort color 1
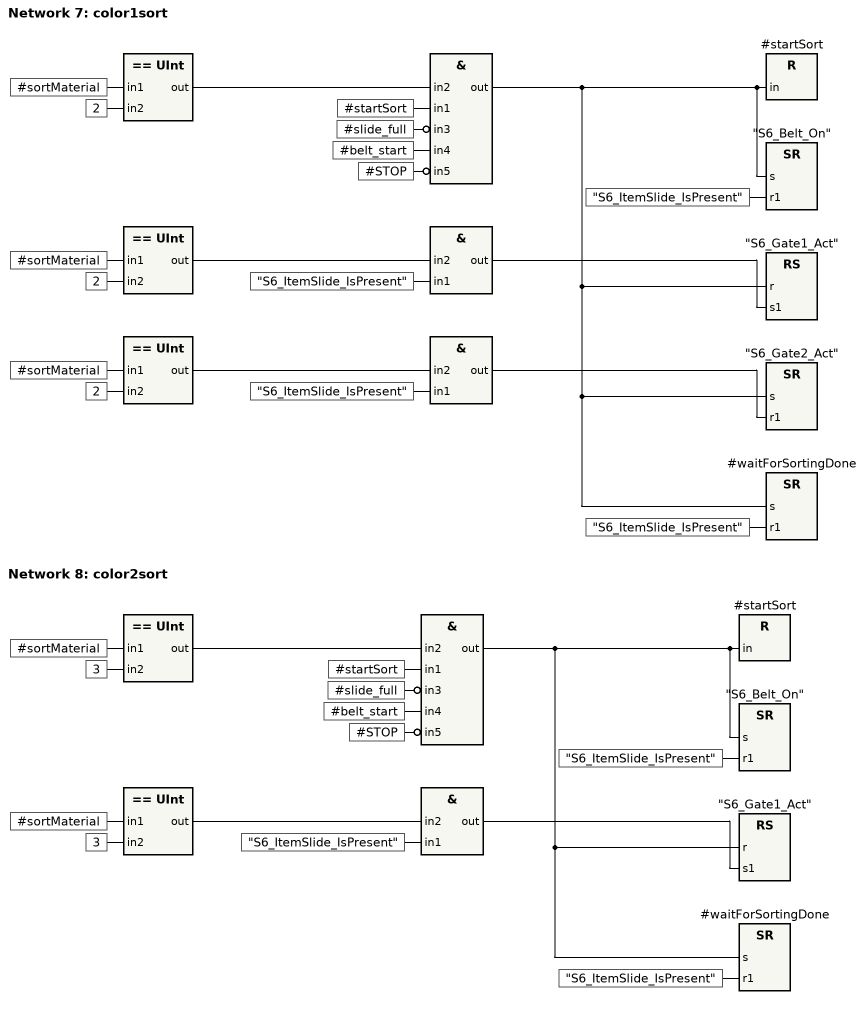
   #_w1 := (#sortMaterial = 2) AND #startSort AND NOT #slide_full AND #belt_start AND NOT #STOP;
   IF #_w1 THEN
       #startSort := FALSE;
       "S6_Belt_On" := TRUE;   // SR flip-flop
   END_IF;
   IF "S6_ItemSlide_IsPresent" THEN "S6_Belt_On" := FALSE; END_IF;
   IF #_w1 THEN
       "S6_Gate1_Act" := FALSE;   // RS flip-flop
   END_IF;
   IF (#sortMaterial = 2) AND "S6_ItemSlide_IsPresent" THEN "S6_Gate1_Act" := TRUE; END_IF;
   IF #_w1 THEN
       "S6_Gate2_Act" := TRUE;   // SR flip-flop
   END_IF;
   IF (#sortMaterial = 2) AND "S6_ItemSlide_IsPresent" THEN "S6_Gate2_Act" := FALSE; END_IF;
   IF #_w1 THEN
       #waitForSortingDone := TRUE;   // SR flip-flop
   END_IF;
   IF "S6_ItemSlide_IsPresent" THEN #waitForSortingDone := FALSE; END_IF;
END_REGION

REGION Network 8: color2sort
   // sort color 2
   #_w1 := (#sortMaterial = 3) AND #startSort AND NOT #slide_full AND #belt_start AND NOT #STOP;
   IF #_w1 THEN
       #startSort := FALSE;
       "S6_Belt_On" := TRUE;   // SR flip-flop
   END_IF;
   IF "S6_ItemSlide_IsPresent" THEN "S6_Belt_On" := FALSE; END_IF;
   IF #_w1 THEN
       "S6_Gate1_Act" := FALSE;   // RS flip-flop
   END_IF;
   IF (#sortMaterial = 3) AND "S6_ItemSlide_IsPresent" THEN "S6_Gate1_Act" := TRUE; END_IF;
   IF #_w1 THEN
       #waitForSortingDone := TRUE;   // SR flip-flop
   END_IF;
   IF "S6_ItemSlide_IsPresent" THEN #waitForSortingDone := FALSE; END_IF;
END_REGION
END_FUNCTION_BLOCK

FUNCTION_BLOCK "Client_interface_target3"   // FB3, FBD
{ S7_Optimized_Access := 'TRUE' }
VERSION : 0.1
   VAR
      connection_done : Bool;
   END_VAR
   VAR_TEMP
      opc_ua_connect_req : Bool;
      opc_ua_connect_done : Bool;
      opc_ua_nsp_done : Bool;
      opc_ua_node_done : Bool;
      opc_ua_rdlist_done : Bool;
   END_VAR
BEGIN

REGION Network 1
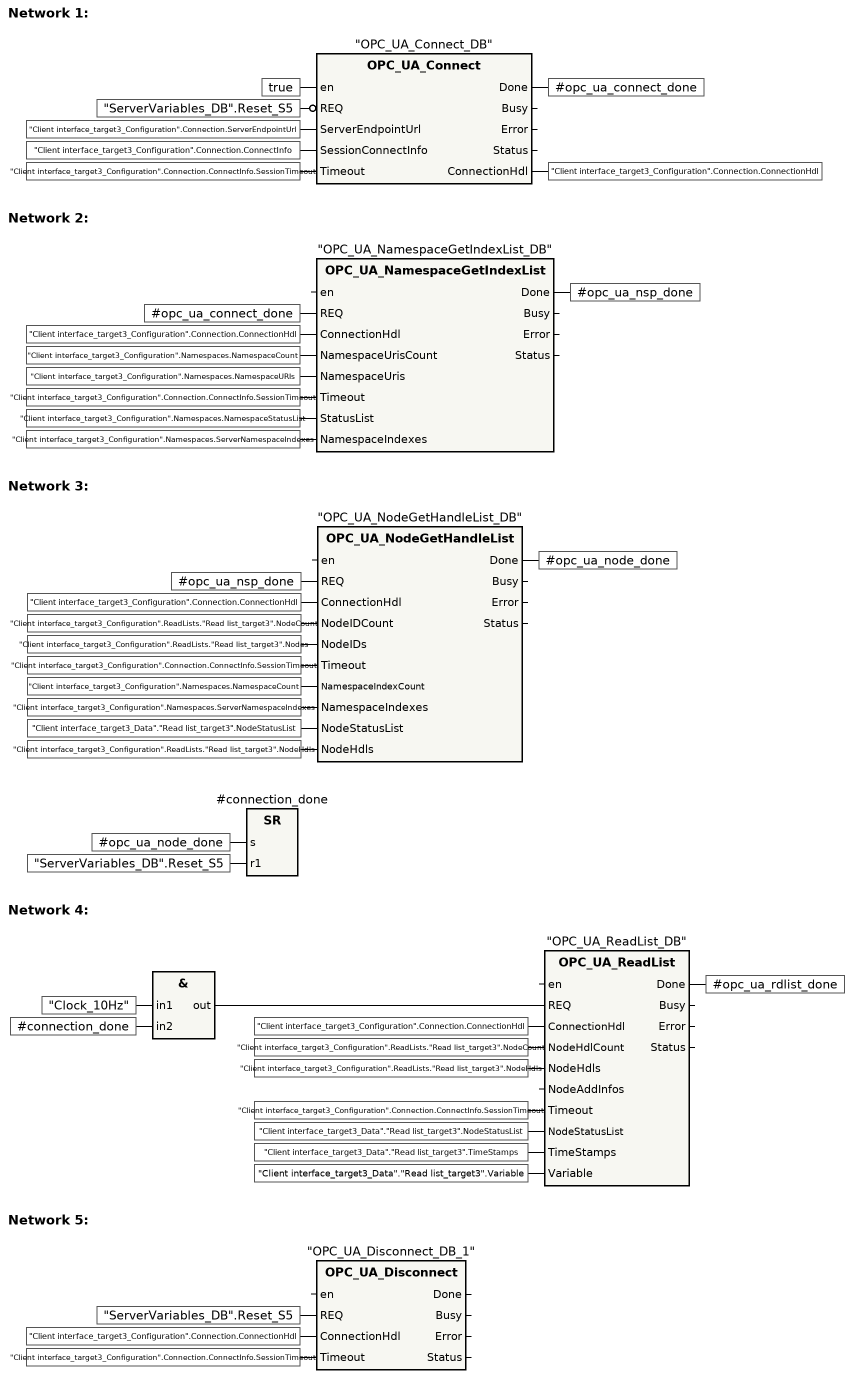
   IF true THEN
       "OPC_UA_Connect_DB"(REQ := NOT "ServerVariables_DB".Reset_S5,   // OPC_UA_Connect
                           ServerEndpointUrl := "Client interface_target3_Configuration".Connection.ServerEndpointUrl,
                           SessionConnectInfo := "Client interface_target3_Configuration".Connection.ConnectInfo,
                           Timeout := "Client interface_target3_Configuration".Connection.ConnectInfo.SessionTimeout,
                           Done => #opc_ua_connect_done,
                           ConnectionHdl => "Client interface_target3_Configuration".Connection.ConnectionHdl);
   END_IF;
END_REGION

REGION Network 2
   "OPC_UA_NamespaceGetIndexList_DB"(REQ := #opc_ua_connect_done,   // OPC_UA_NamespaceGetIndexList
                           ConnectionHdl := "Client interface_target3_Configuration".Connection.ConnectionHdl,
                           NamespaceUrisCount := "Client interface_target3_Configuration".Namespaces.NamespaceCount,
                           NamespaceUris := "Client interface_target3_Configuration".Namespaces.NamespaceURIs,
                           Timeout := "Client interface_target3_Configuration".Connection.ConnectInfo.SessionTimeout,
                           StatusList := "Client interface_target3_Configuration".Namespaces.NamespaceStatusList,
                           NamespaceIndexes := "Client interface_target3_Configuration".Namespaces.ServerNamespaceIndexes,
                           Done => #opc_ua_nsp_done);
END_REGION

REGION Network 3
   "OPC_UA_NodeGetHandleList_DB"(REQ := #opc_ua_nsp_done,   // OPC_UA_NodeGetHandleList
                           ConnectionHdl := "Client interface_target3_Configuration".Connection.ConnectionHdl,
                           NodeIDCount := "Client interface_target3_Configuration".ReadLists."Read list_target3".NodeCount,
                           NodeIDs := "Client interface_target3_Configuration".ReadLists."Read list_target3".Nodes,
                           Timeout := "Client interface_target3_Configuration".Connection.ConnectInfo.SessionTimeout,
                           NamespaceIndexCount := "Client interface_target3_Configuration".Namespaces.NamespaceCount,
                           NamespaceIndexes := "Client interface_target3_Configuration".Namespaces.ServerNamespaceIndexes,
                           NodeStatusList := "Client interface_target3_Data"."Read list_target3".NodeStatusList,
                           NodeHdls := "Client interface_target3_Configuration".ReadLists."Read list_target3".NodeHdls,
                           Done => #opc_ua_node_done);
   IF #opc_ua_node_done THEN
       #connection_done := TRUE;   // SR flip-flop
   END_IF;
   IF "ServerVariables_DB".Reset_S5 THEN #connection_done := FALSE; END_IF;
END_REGION

REGION Network 4
   "OPC_UA_ReadList_DB"(REQ := "Clock_10Hz" AND #connection_done,   // OPC_UA_ReadList
                        ConnectionHdl := "Client interface_target3_Configuration".Connection.ConnectionHdl,
                        NodeHdlCount := "Client interface_target3_Configuration".ReadLists."Read list_target3".NodeCount,
                        NodeHdls := "Client interface_target3_Configuration".ReadLists."Read list_target3".NodeHdls,
                        Timeout := "Client interface_target3_Configuration".Connection.ConnectInfo.SessionTimeout,
                        NodeStatusList := "Client interface_target3_Data"."Read list_target3".NodeStatusList,
                        TimeStamps := "Client interface_target3_Data"."Read list_target3".TimeStamps,
                        Variable := "Client interface_target3_Data"."Read list_target3".Variable,
                        Done => #opc_ua_rdlist_done);
END_REGION

REGION Network 5
   "OPC_UA_Disconnect_DB_1"(REQ := "ServerVariables_DB".Reset_S5,   // OPC_UA_Disconnect
                           ConnectionHdl := "Client interface_target3_Configuration".Connection.ConnectionHdl,
                           Timeout := "Client interface_target3_Configuration".Connection.ConnectInfo.SessionTimeout);
END_REGION
END_FUNCTION_BLOCK

FUNCTION_BLOCK "Client_interface_target1"   // FB4, FBD
{ S7_Optimized_Access := 'TRUE' }
VERSION : 0.1
   VAR
      connection_done : Bool;
   END_VAR
   VAR_TEMP
      opc_ua_connect_done : Bool;
      opc_ua_nsp_done : Bool;
      opc_ua_node_done : Bool;
      opc_ua_rdlist_done : Bool;
   END_VAR
BEGIN

REGION Network 1
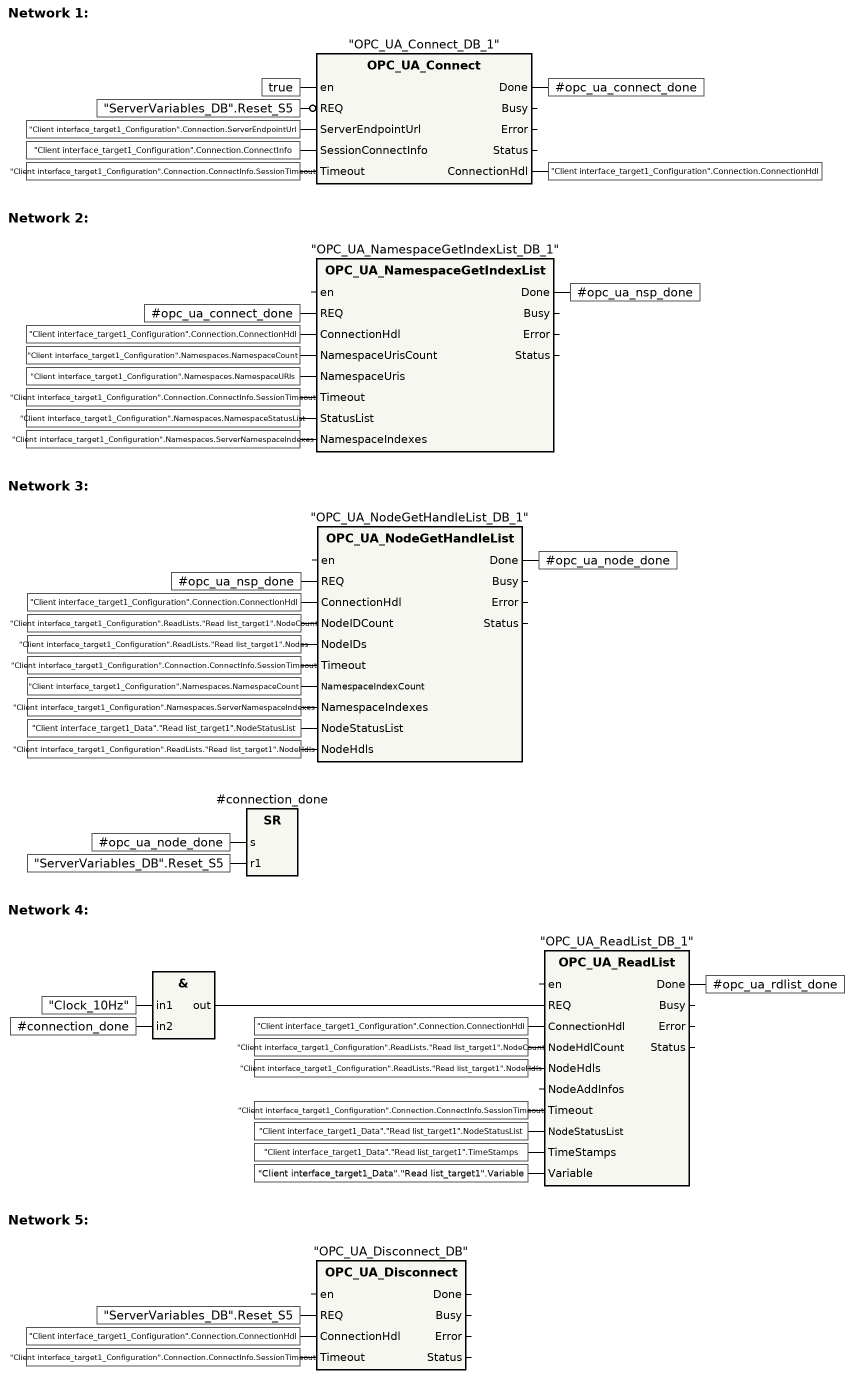
   IF true THEN
       "OPC_UA_Connect_DB_1"(REQ := NOT "ServerVariables_DB".Reset_S5,   // OPC_UA_Connect
                             ServerEndpointUrl := "Client interface_target1_Configuration".Connection.ServerEndpointUrl,
                             SessionConnectInfo := "Client interface_target1_Configuration".Connection.ConnectInfo,
                             Timeout := "Client interface_target1_Configuration".Connection.ConnectInfo.SessionTimeout,
                             Done => #opc_ua_connect_done,
                             ConnectionHdl => "Client interface_target1_Configuration".Connection.ConnectionHdl);
   END_IF;
END_REGION

REGION Network 2
   "OPC_UA_NamespaceGetIndexList_DB_1"(REQ := #opc_ua_connect_done,   // OPC_UA_NamespaceGetIndexList
                           ConnectionHdl := "Client interface_target1_Configuration".Connection.ConnectionHdl,
                           NamespaceUrisCount := "Client interface_target1_Configuration".Namespaces.NamespaceCount,
                           NamespaceUris := "Client interface_target1_Configuration".Namespaces.NamespaceURIs,
                           Timeout := "Client interface_target1_Configuration".Connection.ConnectInfo.SessionTimeout,
                           StatusList := "Client interface_target1_Configuration".Namespaces.NamespaceStatusList,
                           NamespaceIndexes := "Client interface_target1_Configuration".Namespaces.ServerNamespaceIndexes,
                           Done => #opc_ua_nsp_done);
END_REGION

REGION Network 3
   "OPC_UA_NodeGetHandleList_DB_1"(REQ := #opc_ua_nsp_done,   // OPC_UA_NodeGetHandleList
                           ConnectionHdl := "Client interface_target1_Configuration".Connection.ConnectionHdl,
                           NodeIDCount := "Client interface_target1_Configuration".ReadLists."Read list_target1".NodeCount,
                           NodeIDs := "Client interface_target1_Configuration".ReadLists."Read list_target1".Nodes,
                           Timeout := "Client interface_target1_Configuration".Connection.ConnectInfo.SessionTimeout,
                           NamespaceIndexCount := "Client interface_target1_Configuration".Namespaces.NamespaceCount,
                           NamespaceIndexes := "Client interface_target1_Configuration".Namespaces.ServerNamespaceIndexes,
                           NodeStatusList := "Client interface_target1_Data"."Read list_target1".NodeStatusList,
                           NodeHdls := "Client interface_target1_Configuration".ReadLists."Read list_target1".NodeHdls,
                           Done => #opc_ua_node_done);
   IF #opc_ua_node_done THEN
       #connection_done := TRUE;   // SR flip-flop
   END_IF;
   IF "ServerVariables_DB".Reset_S5 THEN #connection_done := FALSE; END_IF;
END_REGION

REGION Network 4
   "OPC_UA_ReadList_DB_1"(REQ := "Clock_10Hz" AND #connection_done,   // OPC_UA_ReadList
                          ConnectionHdl := "Client interface_target1_Configuration".Connection.ConnectionHdl,
                          NodeHdlCount := "Client interface_target1_Configuration".ReadLists."Read list_target1".NodeCount,
                          NodeHdls := "Client interface_target1_Configuration".ReadLists."Read list_target1".NodeHdls,
                          Timeout := "Client interface_target1_Configuration".Connection.ConnectInfo.SessionTimeout,
                          NodeStatusList := "Client interface_target1_Data"."Read list_target1".NodeStatusList,
                          TimeStamps := "Client interface_target1_Data"."Read list_target1".TimeStamps,
                          Variable := "Client interface_target1_Data"."Read list_target1".Variable,
                          Done => #opc_ua_rdlist_done);
END_REGION

REGION Network 5
   "OPC_UA_Disconnect_DB"(REQ := "ServerVariables_DB".Reset_S5,   // OPC_UA_Disconnect
                          ConnectionHdl := "Client interface_target1_Configuration".Connection.ConnectionHdl,
                          Timeout := "Client interface_target1_Configuration".Connection.ConnectInfo.SessionTimeout);
END_REGION
END_FUNCTION_BLOCK

FUNCTION_BLOCK "FIFO"   // FB5, FBD
{ S7_Optimized_Access := 'TRUE' }
VERSION : 0.1
// FIFO with 4 elements. first element fans out
   VAR_INPUT
      read : Bool;
      write : Bool;
      data_in : UInt;
      reset : Bool;
   END_VAR
   VAR_OUTPUT
      data_out : UInt;
      full : Bool;
      empty : Bool;
   END_VAR
   VAR
      read_pos : UInt;
      write_pos : UInt;
      fill_count : UInt := 0;
      data0 : UInt;
      data1 : UInt;
      data2 : UInt;
      data3 : UInt;
      write_occured : Bool;
      read_occured : Bool;
      trigger : Bool;
      waitForNegWrite : Bool;
      waitForNegRead : Bool;
   END_VAR
BEGIN

REGION Network 1: reset
   // reset the values of the fifo buffer (read and write positions)
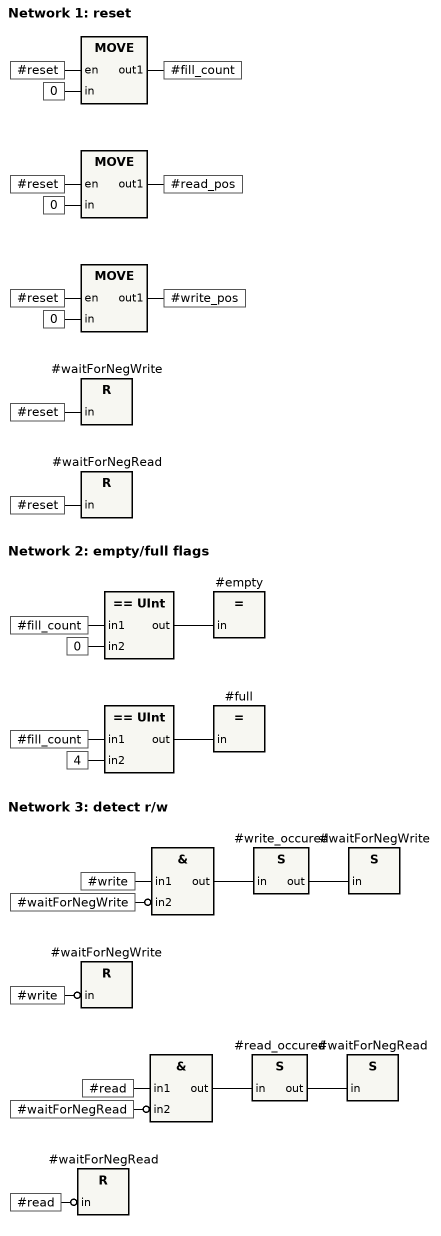
   IF #reset THEN
       #fill_count := 0;
       #read_pos := 0;
       #write_pos := 0;
       #waitForNegWrite := FALSE;
       #waitForNegRead := FALSE;
   END_IF;
END_REGION

REGION Network 2: empty/full flags
   // set a specific full/empty flag when buffer is full or contains no actual item (material info)
   #empty := #fill_count = 0;
   #full := #fill_count = 4;
END_REGION

REGION Network 3: detect r/w
   // detect if a read or write input boolean flag will be high
   IF #write AND NOT #waitForNegWrite THEN
       #write_occured := TRUE;
       #waitForNegWrite := TRUE;
   END_IF;
   IF NOT #write THEN #waitForNegWrite := FALSE; END_IF;
   IF #read AND NOT #waitForNegRead THEN
       #read_occured := TRUE;
       #waitForNegRead := TRUE;
   END_IF;
   IF NOT #read THEN #waitForNegRead := FALSE; END_IF;
END_REGION

REGION Network 4: data out logic
   // always output data of current read_pos
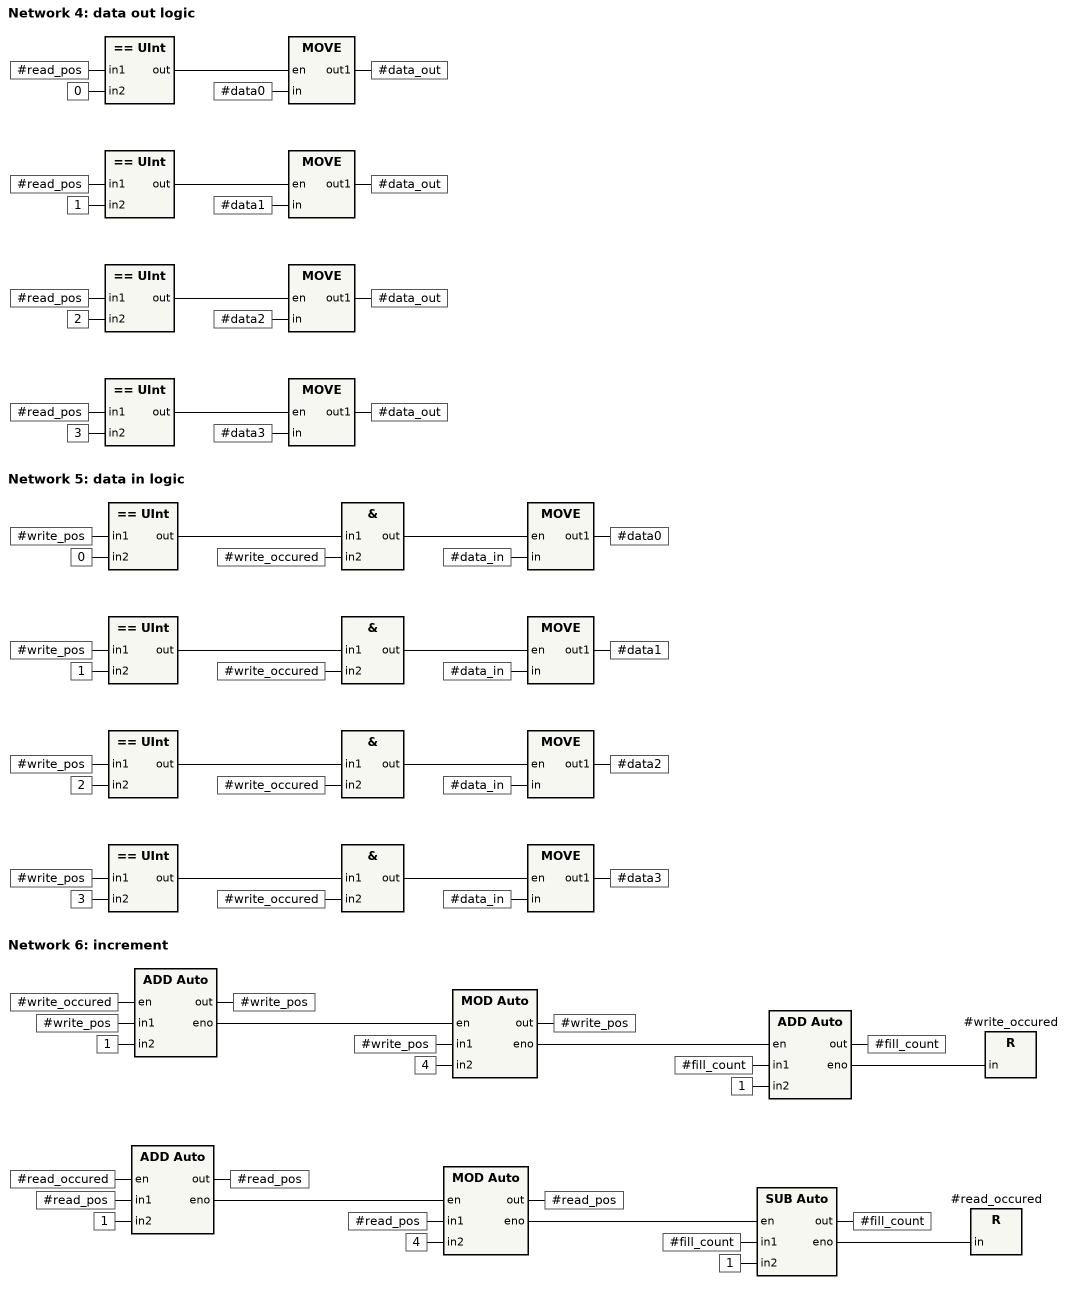
   IF #read_pos = 0 THEN #data_out := #data0; END_IF;
   IF #read_pos = 1 THEN #data_out := #data1; END_IF;
   IF #read_pos = 2 THEN #data_out := #data2; END_IF;
   IF #read_pos = 3 THEN #data_out := #data3; END_IF;
END_REGION

REGION Network 5: data in logic
   // set the correct data regarding the write position when a write occured on the input
   IF (#write_pos = 0) AND #write_occured THEN #data0 := #data_in; END_IF;
   IF (#write_pos = 1) AND #write_occured THEN #data1 := #data_in; END_IF;
   IF (#write_pos = 2) AND #write_occured THEN #data2 := #data_in; END_IF;
   IF (#write_pos = 3) AND #write_occured THEN #data3 := #data_in; END_IF;
END_REGION

REGION Network 6: increment
   // Set the correct read and write positions
   IF #write_occured THEN
       #write_pos := #write_pos + 1;
       #write_pos := #write_pos MOD 4;
       #fill_count := #fill_count + 1;
       #write_occured := FALSE;
   END_IF;
   IF #read_occured THEN
       #read_pos := #read_pos + 1;
       #read_pos := #read_pos MOD 4;
       #fill_count := #fill_count - 1;
       #read_occured := FALSE;
   END_IF;
END_REGION

REGION Network 7: reset occurence
   // reset occurence variables
END_REGION
END_FUNCTION_BLOCK

ORGANIZATION_BLOCK "Main"   // OB1, LAD, ProgramCycle
TITLE = "Main Program Sweep (Cycle)"
{ S7_Optimized_Access := 'TRUE' }
VERSION : 0.1
   VAR_INPUT
      Initial_Call : Bool;   // Initial call of this OB
      Remanence : Bool;   // =True, if remanent data are available
   END_VAR
   VAR_TEMP
      global_error_56 : Bool;
      station4_req : Bool;
      station6_sorting_done : Bool;
      station5_ack : Bool;
      global_error : Bool;
      station4_material_info : Int;
      station6_slidefull : Bool;
      station6_ack : Bool;
      station5_req : Bool;
      material : Int;
      belt_start : Bool;
   END_VAR
BEGIN

REGION Network 1: Initial call of this OB
   // still the buttons have to be modelled for the user
   // added variables from plc tags of station5: 
   // - 'ack' as acknowledge from station5 to 4
   // - 'request' as request from station 4 to 5 --> workpiece ready
   // - 'material' as Uint that keeps info about red, black and silver workpieces
   // - emergency_stop: a global error occured on the plant
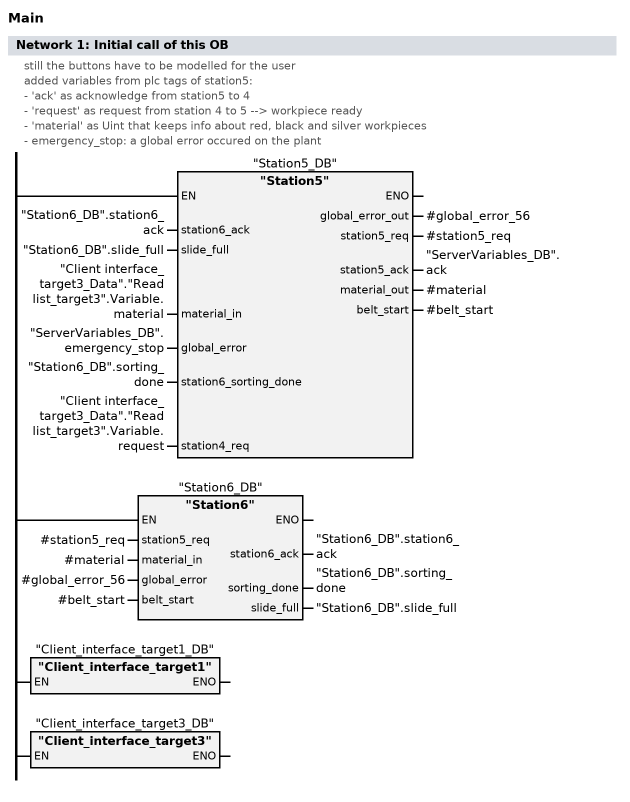
   RUNG wire#powerrail
      "Station5_DB"(station6_ack := "Station6_DB".station6_ack, slide_full := "Station6_DB".slide_full, material_in := "Client interface_target3_Data"."Read list_target3".Variable.material, global_error := "ServerVariables_DB".emergency_stop, station6_sorting_done := "Station6_DB".sorting_done, station4_req := "Client interface_target3_Data"."Read list_target3".Variable.request, global_error_out => #global_error_56, station5_req => #station5_req, station5_ack => "ServerVariables_DB".ack, material_out => #material, belt_start => #belt_start)
   END_RUNG
   RUNG wire#powerrail
      "Station6_DB"(station5_req := #station5_req, material_in := #material, global_error := #global_error_56, belt_start := #belt_start, station6_ack => "Station6_DB".station6_ack, sorting_done => "Station6_DB".sorting_done, slide_full => "Station6_DB".slide_full)
   END_RUNG
   RUNG wire#powerrail
      "Client_interface_target1_DB"()
   END_RUNG
   RUNG wire#powerrail
      "Client_interface_target3_DB"()
   END_RUNG
   // the same network as SCL:
   "Station5_DB"(station6_ack := "Station6_DB".station6_ack,   // "Station5"
                 slide_full := "Station6_DB".slide_full,
                 material_in := "Client interface_target3_Data"."Read list_target3".Variable.material,
                 global_error := "ServerVariables_DB".emergency_stop,
                 station6_sorting_done := "Station6_DB".sorting_done,
                 station4_req := "Client interface_target3_Data"."Read list_target3".Variable.request,
                 global_error_out => #global_error_56,
                 station5_req => #station5_req,
                 station5_ack => "ServerVariables_DB".ack,
                 material_out => #material,
                 belt_start => #belt_start);
   "Station6_DB"(station5_req := #station5_req,   // "Station6"
                 material_in := #material,
                 global_error := #global_error_56,
                 belt_start := #belt_start,
                 station6_ack => "Station6_DB".station6_ack,
                 sorting_done => "Station6_DB".sorting_done,
                 slide_full => "Station6_DB".slide_full);
   "Client_interface_target1_DB"();   // "Client_interface_target1"
   "Client_interface_target3_DB"();   // "Client_interface_target3"
END_REGION
END_ORGANIZATION_BLOCK

(* ===== HMI "HMI_RT_1" =====
system functions are stored by id; their names below are inferred from use
connection "HMI_Connection_1": ETHERNET, S7_1500_OMS

HMI tags "Default tag table"
   "Tag_ScreenNumber" : UInt, internal

screen "Root screen" 1280x740, template "Template_1"
   on GenerateScreen: SetTag("Tag_ScreenNumber", 1)
   TextField "HmiScreenItemData" at 128,90 size 1024x27; Text 'Welcome to HMI_1 (TP1500 Comfort V2)!'
   Clock "Clock_1" at 0,172 size 1280x466

Template "Template_1" 1280x740
   Button "Exit" at 1200,679 size 78x59; TextOff 'Exit'; PictureOff "ExitRuntime_TP1500_Comfort_V2_TR"; PictureOn "ExitRuntime_TP1500_Comfort_V2_TR"
      on Release: StopRuntime(0)
   Button "Template_Button" at 1120,679 size 78x59; TextOff 'Text'
   Button "Template_Button_1" at 1040,679 size 78x59; TextOff 'Text'
   Button "Template_Button_2" at 960,679 size 78x59; TextOff 'Text'
   Button "Template_Button_3" at 880,679 size 78x59; TextOff 'Text'
   Button "Template_Button_4" at 800,679 size 78x59; TextOff 'Text'
   Button "Template_Button_5" at 720,679 size 78x59; TextOff 'Text'
   Button "Template_Button_6" at 640,679 size 78x59; TextOff 'Text'
   Button "Template_Button_7" at 561,679 size 78x59; TextOff 'Text'
   Button "Template_Button_8" at 481,679 size 78x59; TextOff 'Text'
   Button "Template_Button_9" at 401,679 size 78x59; TextOff 'Text'
   Button "Template_Button_10" at 321,679 size 78x59; TextOff 'Text'
   Button "Template_Button_11" at 241,679 size 78x59; TextOff 'Text'
   Button "Template_Button_12" at 161,679 size 78x59; TextOff 'Text'
   Button "Template_Button_13" at 81,679 size 78x59; TextOff 'Text'
   Button "Start screen" at 1,679 size 78x59; TextOff 'Start screen'; PictureOff "NavigateHome_TP1500_Comfort_V2_TR"; PictureOn "NavigateHome_TP1500_Comfort_V2_TR"
      on Release: ActivateScreen("Root screen", 0)
*)